{attribute 'qualified_only'}
{attribute 'strict'}
TYPE E_ControlModeSP :
(
    ManualControl := 2,
    CloseValve := 3,
    OpenValve := 4,
    PressureControl := 5,
    HoldValve := 6,
    LearnProcedure := 7
) USINT := CloseValve;
END_TYPE

(* stored: Version 1.1.0.1
   DUT E_ControlModeSP: Id {ba6b9899-bb05-401a-88ad-c50fd12e5d8e} *)
